    if not set_grind_process_state(True, pattern_circle(circle_diam_m, n_cycles, True)):
      return False
    end

    # Grind the pattern
    imover_realtime(False) # True seems to workl!?
    start_user_timer()
    pattern_circle(circle_diam_m, n_cycles)
    stop_user_timer()

    if not stay_in_contact or not ok_to_proceed():
      set_grind_process_state(False)
    end
    return True

    if grind_linear_blend_radius_m > 0.0:
      # Try setting n_sides to 1.5 blend radii
      local circum_m = MATH_PI * circle_diam_mm / 1000.
      global grind_circle_n_sides = ceil(circum_m / (grind_linear_blend_radius_m * 1.5))
    end

    return grind_poly(circle_diam_mm, grind_circle_n_sides, n_cycles, stay_in_contact)
  end

  # Grind along a circle with circle_diam_m. Repeat n_cycles times.
  # If return_initial_offset_only, just returns dp to initial drawing point
  def pattern_circle(circle_diam_m, n_cycles, return_initial_offset_only = False):
    local circle_radius_m = circle_diam_m / 2.0
    local n_points = recommend_npoints(circle_diam_m, grind_linear_vel_mps)

    local dp1 = p[-circle_radius_m, 0, 0, 0, 0, 0]
    if return_initial_offset_only:
      return dp1
    end

    global grind_cycle = 1
    while (ok_to_proceed() and grind_cycle <= n_cycles):
      socket_send_number("grind_cycle", grind_cycle)
      local i = 0
      while ok_to_proceed() and i <= n_points:
        local theta = d2r(180.0 + 360.0 * i / n_points)
        local x = circle_radius_m * cos(theta)
        local y = circle_radius_m * sin(theta)

        local dc = [x, y, 0]
        if not ok_to_proceed() or i == n_points:
          drawgi_finish(dc)
        else:
          drawgi_to(dc)
        end
        i = i + 1
      end

      grind_cycle = grind_cycle + 1
    end

    return dp1
  end

  # Grind along a spiral circle1_diam_mm to circle2_diam_mm in n_revolutions with rotations centered on current tool position. Repeat n_cycles times. If stay_in_contact, stay_in_contact at end.
  def grind_spiral(circle1_diam_mm, circle2_diam_mm, n_revolutions, n_cycles, stay_in_contact):
    if n_cycles < 1:
      return True
    end

    local circle1_diam_m = circle1_diam_mm / 1000.0
    local circle2_diam_m = circle2_diam_mm / 1000.0
    local part_diam_m = robot_part_geometry[1] / 1000.0

    # Grind time estimate based on average diam
    local avg_diam_mm = (circle1_diam_mm + circle2_diam_mm) / 2.0
    local time_ms = MATH_PI * avg_diam_mm * n_revolutions * n_cycles / grind_linear_vel_mps + 1500
    socket_send_number("robot_step_time_estimate_ms", time_ms)

    if not set_grind_process_state(True, pattern_spiral(circle1_diam_m, circle2_diam_m, n_revolutions, n_cycles, True)):
      return False
    end

    # Grind the pattern
    imover_realtime(False) # True fails!?
    start_user_timer()
    pattern_spiral(circle1_diam_m, circle2_diam_m, n_revolutions, n_cycles)
    stop_user_timer()

    if not stay_in_contact or not ok_to_proceed():
      set_grind_process_state(False)
    end

    return True
  end

  # Grind a spiral from diam1 to diam2 in n_revolutions revolutions. Repeat n_cycles times.
  # If return_initial_offset_only, just returns dp to initial drawing point
  def pattern_spiral(circle1_diam_m, circle2_diam_m, n_revolutions, n_cycles, return_initial_offset_only = False):
    local max_diam_m = max(circle1_diam_m, circle2_diam_m)
    local circle1_radius_m = circle1_diam_m / 2.0
    local circle2_radius_m = circle2_diam_m / 2.0

    local dp1 = p[-circle1_radius_m, 0, 0, 0, 0, 0]
    if return_initial_offset_only:
      return dp1
    end

    global grind_cycle = 1
    while (ok_to_proceed() and grind_cycle <= n_cycles):
      socket_send_number("grind_cycle", grind_cycle)

      # Initial conditions
      local theta = d2r(180.0)
      local r_m = circle1_radius_m
      local revs_completed = 0.0
      local rev_slope = (circle2_radius_m - circle1_radius_m) / n_revolutions
      local move_m = grind_linear_blend_radius_m * 2

      while ok_to_proceed() and revs_completed < n_revolutions:
        local delta_theta = move_m / r_m
        local theta = theta + delta_theta
        local x = r_m * cos(theta)
        local y = r_m * sin(theta)

        local dc = [x, y, 0]
        if not ok_to_proceed() or revs_completed >= n_revolutions:
          drawgi_finish(dc)
        else:
          drawgi_to(dc)
        end

        local revs_completed = revs_completed + delta_theta / (2 * MATH_PI)
        local r_m = circle1_radius_m + rev_slope * revs_completed
      end

      grind_cycle = grind_cycle + 1

      # Next cycle- swap diameters so we go in/out/in etc.
      local old_circle1_radius_m = circle1_radius_m
      local circle1_radius_m = circle2_radius_m
      local circle2_radius_m = old_circle1_radius_m
    end

    return dp1
  end
  #
  # END TOP LEVEL GRIND FUNCTIONS AND THEIR PATTERNS
  ######################################################################################
  $ 5 "init_autogrind()"
  init_autogrind()
  $ 6 "currentTcpPose≔get_actual_tcp_pose()"
  global currentTcpPose= get_actual_tcp_pose ()
  $ 7 "MoveJ"
  $ 8 "currentTcpPose" "breakAfter"
  movej(currentTcpPose, a=1.3962634015954636, v=1.0471975511965976)
  $ 9 "socket_is_open≔ False "
  global socket_is_open=  False
  while (True):
    $ 10 "Robot Program"
    $ 11 "Loop socket_is_open ≟  False "
    while (socket_is_open  ==    False  ):
      $ 12 "Wait: 0.25"
      sleep(0.25)
      $ 13 "socket_close()"
      socket_close()
      $ 14 "socket_is_open≔socket_open('169.254.254.200', 30000)"
      global socket_is_open=socket_open("169.254.254.200", 30000)
      $ 15 "If not socket_is_open"
      if (not socket_is_open):
        $ 16 "socket_is_open≔socket_open('169.254.254.210', 30000)"
        global socket_is_open=socket_open("169.254.254.210", 30000)
      end
      $ 17 "If not socket_is_open"
      if (not socket_is_open):
        $ 18 "socket_is_open≔socket_open('192.168.0.252', 30000)"
        global socket_is_open=socket_open("192.168.0.252", 30000)
      end
    end
    $ 19 "response≔'Unknown command'"
    global response="Unknown command"
    $ 20 "command≔socket_read_ascii_float(12)"
    global command=socket_read_ascii_float(12)
    $ 21 "If command_validate()"
    if (command_validate()):
      $ 22 "command_start()"
      command_start()
      $ 23 "Set Stacklight=On"
      set_standard_digital_out(0, True)
      $ 24 "Switch command[1]"
      switch_1 = command[1]
      $ 25 "Case 10"
      if (10 == switch_1):
        $ 26 "return_actual_tcp_pose()"
        return_actual_tcp_pose()
      elif (12 == switch_1):
        $ 27 "Case 12"
        $ 28 "return_tcp_offset()"
        return_tcp_offset()
      elif (13 == switch_1):
        $ 29 "Case 13"
        $ 30 "movel_relative_base(p[command[2], command[3], command[4], command[5], command[6], command[7]])"
        movel_relative_base(p[command[2], command[3], command[4], command[5], command[6], command[7]])
      elif (14 == switch_1):
        $ 31 "Case 14"
        $ 32 "movel_relative_tcp(p[command[2], command[3], command[4], command[5], command[6], command[7]])"
        movel_relative_tcp(p[command[2], command[3], command[4], command[5], command[6], command[7]])
      elif (15 == switch_1):
        $ 33 "Case 15"
        $ 34 "movel_relative_tcp_part(p[command[2], command[3], command[4], command[5], command[6], command[7]])"
        movel_relative_tcp_part(p[command[2], command[3], command[4], command[5], command[6], command[7]])
      elif (16 == switch_1):
        $ 35 "Case 16"
        $ 36 "movel_one_only(command[2],command[3])"
        movel_one_only(command[2],command[3])
      elif (18 == switch_1):
        $ 37 "Case 18"
        $ 38 "movel_rot_only(command[2],command[3],command[4])"
        movel_rot_only(command[2],command[3],command[4])
      elif (20 == switch_1):
        $ 39 "Case 20"
        $ 40 "return_get_actual_joint_positions()"
        return_get_actual_joint_positions()
      elif (21 == switch_1):
        $ 41 "Case 21"
        $ 42 "movej_ag([command[2], command[3], command[4], command[5], command[6], command[7]])"
        movej_ag([command[2], command[3], command[4], command[5], command[6], command[7]])
      elif (22 == switch_1):
        $ 43 "Case 22"
        $ 44 "movel_ag(p[command[2], command[3], command[4], command[5], command[6], command[7]])"
        movel_ag(p[command[2], command[3], command[4], command[5], command[6], command[7]])
      elif (25 == switch_1):
        $ 45 "Case 25"
        $ 46 "return_both_positions()"
        return_both_positions()
      elif (30 == switch_1):
        $ 47 "Case 30"
        $ 48 "set_variable()"
        set_variable()
      elif (35 == switch_1):
        $ 49 "Case 35"
        $ 50 "set_grind_variable()"
        set_grind_variable()
      elif (40 == switch_1):
        $ 51 "Case 40"
        $ 52 "grind()"
        grind()
      elif (98 == switch_1):
        $ 53 "Case 98"
        $ 54 "response≔'socket reset'"
        global response="socket reset"
      elif (99 == switch_1):
        $ 55 "Case 99"
        $ 56 "response≔'exiting'"
        global response="exiting"
      else:
        $ 57 "Default Case"
        $ 58 "response≔'unknown command'"
        global response="unknown command"
      end
      $ 59 "command_finish()"
      command_finish()
      $ 60 "Set Stacklight=Off"
      set_standard_digital_out(0, False)
      $ 61 "If command[1]≟98"
      if (command[1] == 98):
        $ 62 "Wait: 0.5"
        sleep(0.5)
        $ 63 "socket_close()"
        socket_close()
        $ 64 "socket_is_open≔ False "
        global socket_is_open=  False
      end
      $ 65 "If command[1]≟99"
      if (command[1] == 99):
        $ 66 "Wait: 0.5"
        sleep(0.5)
        $ 67 "socket_close()"
        socket_close()
        $ 68 "socket_is_open≔ False "
        global socket_is_open=  False
        $ 69 "Halt"
        halt
      end
    else:
      $ 70 "Else" "noBreak"
      $ 71 "no_command()"
      no_command()
    end
  end
end
